// Tests for AstroBROT.FB_RADEC2HADEC (ICRS RA/Dec -> apparent hour angle / Dec; the block IAG50cm uses).
//
// GENERATED by AstroBROT/testing/gen_block_tests.py from testing/golden_blocks.py, do not edit the numbers by hand.
// Every golden case is checked against the Python port of the ST (1E-7 deg) and against erfa.atco13 as a great-circle
// separation on the (HA, Dec) sphere (2E-4 deg = 0.72 arcsec; the port is 0.2 to 0.4 arcsec away, mostly the diurnal
// aberration that the ST leaves out). The dut1 shift itself is also covered in FB_DUT1_Tests.
//
// Every call assigns all inputs: FB_RADEC2HADEC still writes its precessed and corrected position back into ra and dec
// (issue #8), so these tests must not rely on ra / dec surviving a call.
FUNCTION_BLOCK FB_RADEC2HADEC_Tests EXTENDS TcUnit.FB_TestSuite
VAR
END_VAR

Golden_Tenerife_2026();
Golden_Tenerife_low();
Golden_South_2010();
Golden_Dut1();
Golden_RA_Wrap();
Golden_Poles();
Golden_Near_The_Poles();
Right_Ascension_Is_Periodic();
Longitude_Is_Periodic();
Outputs_Stay_In_Range();
Time_Inputs_Are_Not_Modified();

METHOD PRIVATE CheckNear
VAR_INPUT
	fExpected	: LREAL;
	fActual	: LREAL;
	fDelta	: LREAL;
	sName	: STRING(255);
END_VAR
AssertEquals_LREAL(Expected := fExpected, Actual := fActual, Delta := fDelta, Message := sName);
END_METHOD

METHOD PRIVATE CheckAngle
VAR_INPUT
	fExpected	: LREAL;
	fActual	: LREAL;
	fDelta	: LREAL;
	sName	: STRING(255);
END_VAR
VAR
	fDiff	: LREAL;
END_VAR
// angles in degrees, compared modulo 360 so that 359.9999999 and -1.0E-7 are equal
fDiff := fActual - fExpected;
WHILE fDiff > 180.0 DO fDiff := fDiff - 360.0; END_WHILE
WHILE fDiff < -180.0 DO fDiff := fDiff + 360.0; END_WHILE
AssertEquals_LREAL(Expected := 0.0, Actual := fDiff, Delta := fDelta, Message := sName);
END_METHOD

METHOD PRIVATE CheckSeparation
VAR_INPUT
	fLon1	: LREAL;
	fLat1	: LREAL;
	fLon2	: LREAL;
	fLat2	: LREAL;
	fDelta	: LREAL;
	sName	: STRING(255);
END_VAR
VAR
	fD2r	: LREAL;
	fHalfDLat	: LREAL;
	fHalfDLon	: LREAL;
	fHav	: LREAL;
	fSep	: LREAL;
END_VAR
// great-circle separation of two positions (longitude, latitude in degrees) against a tolerance in degrees;
// a difference of longitudes is not a distance on the sky, this is (haversine formula)
fD2r := 0.017453292519943295;
fHalfDLat := (fLat2 - fLat1) * fD2r * 0.5;
fHalfDLon := (fLon2 - fLon1) * fD2r * 0.5;
fHav := SIN(fHalfDLat) * SIN(fHalfDLat) + COS(fLat1 * fD2r) * COS(fLat2 * fD2r) * SIN(fHalfDLon) * SIN(fHalfDLon);
fSep := 2.0 * ASIN(SQRT(LIMIT(0.0, fHav, 1.0))) / fD2r;
AssertEquals_LREAL(Expected := 0.0, Actual := fSep, Delta := fDelta, Message := sName);
END_METHOD

METHOD PRIVATE Golden_Tenerife_2026
VAR
	fb	: AstroBROT.FB_RADEC2HADEC;
END_VAR
TEST('Golden_Tenerife_2026');
fb(jd := 2461300.75, ra := 83.63, dec := 22.01, lon := -16.5, dut1 := 0.0);
CheckAngle(345.6575630310487, fb.ha_out, 1.0E-7, 'Tenerife_2026 ha');
CheckNear(22.02849232968123, fb.dec_out, 1.0E-7, 'Tenerife_2026 dec');
CheckSeparation(345.65746144326204, 22.028485286326138, fb.ha_out, fb.dec_out, 0.0002, 'Tenerife_2026 vs erfa');
TEST_FINISHED();
END_METHOD

METHOD PRIVATE Golden_Tenerife_low
VAR
	fb	: AstroBROT.FB_RADEC2HADEC;
END_VAR
TEST('Golden_Tenerife_low');
fb(jd := 2461300.75, ra := 130.0, dec := -10.0, lon := -16.5, dut1 := 0.0);
CheckAngle(299.37201176540054, fb.ha_out, 1.0E-7, 'Tenerife_low ha');
CheckNear(-10.091922210560911, fb.dec_out, 1.0E-7, 'Tenerife_low dec');
CheckSeparation(299.3719555337581, -10.091909866750818, fb.ha_out, fb.dec_out, 0.0002, 'Tenerife_low vs erfa');
TEST_FINISHED();
END_METHOD

METHOD PRIVATE Golden_South_2010
VAR
	fb	: AstroBROT.FB_RADEC2HADEC;
END_VAR
TEST('Golden_South_2010');
fb(jd := 2455197.5, ra := 312.5, dec := -47.3, lon := -70.7, dut1 := 0.0);
CheckAngle(77.17023586398261, fb.ha_out, 1.0E-7, 'South_2010 ha');
CheckNear(-47.26426875549772, fb.dec_out, 1.0E-7, 'South_2010 dec');
CheckSeparation(77.17019695311718, -47.26432489859199, fb.ha_out, fb.dec_out, 0.0002, 'South_2010 vs erfa');
TEST_FINISHED();
END_METHOD

METHOD PRIVATE Golden_Dut1
VAR
	fb	: AstroBROT.FB_RADEC2HADEC;
END_VAR
TEST('Golden_Dut1');
fb(jd := 2461300.75, ra := 83.63, dec := 22.01, lon := -16.5, dut1 := 0.9);
CheckAngle(345.6613233618934, fb.ha_out, 1.0E-7, 'Tenerife_dut1_plus ha');
CheckNear(22.02849232968123, fb.dec_out, 1.0E-7, 'Tenerife_dut1_plus dec');
CheckSeparation(345.66122170868215, 22.028485288193934, fb.ha_out, fb.dec_out, 0.0002, 'Tenerife_dut1_plus vs erfa');
fb(jd := 2461300.75, ra := 83.63, dec := 22.01, lon := -16.5, dut1 := -0.9);
CheckAngle(345.65380270020404, fb.ha_out, 1.0E-7, 'Tenerife_dut1_minus ha');
CheckNear(22.02849232968123, fb.dec_out, 1.0E-7, 'Tenerife_dut1_minus dec');
CheckSeparation(345.653701177839, 22.028485284458373, fb.ha_out, fb.dec_out, 0.0002, 'Tenerife_dut1_minus vs erfa');
TEST_FINISHED();
END_METHOD

METHOD PRIVATE Golden_RA_Wrap
VAR
	fb	: AstroBROT.FB_RADEC2HADEC;
END_VAR
TEST('Golden_RA_Wrap');
fb(jd := 2461300.75, ra := 0.0001, dec := 22.01, lon := -16.5, dut1 := 0.0);
CheckAngle(69.34278166497118, fb.ha_out, 1.0E-7, 'RA_wrap_low ha');
CheckNear(22.16156103752678, fb.dec_out, 1.0E-7, 'RA_wrap_low dec');
CheckSeparation(69.34272927043514, 22.16158906186533, fb.ha_out, fb.dec_out, 0.0002, 'RA_wrap_low vs erfa');
fb(jd := 2461300.75, ra := 359.9999, dec := 22.01, lon := -16.5, dut1 := 0.0);
CheckAngle(69.34298187519398, fb.ha_out, 1.0E-7, 'RA_wrap_high ha');
CheckNear(22.16156103790214, fb.dec_out, 1.0E-7, 'RA_wrap_high dec');
CheckSeparation(69.34292948093092, 22.161589062278132, fb.ha_out, fb.dec_out, 0.0002, 'RA_wrap_high vs erfa');
TEST_FINISHED();
END_METHOD

METHOD PRIVATE Golden_Poles
VAR
	fb	: AstroBROT.FB_RADEC2HADEC;
END_VAR
TEST('Golden_Poles');
fb(jd := 2461300.75, ra := 0.0, dec := 90.0, lon := -16.5, dut1 := 0.0);
CheckAngle(250.63644034864151, fb.ha_out, 1.0E-7, 'North_pole ha');
CheckNear(89.85080571177119, fb.dec_out, 1.0E-7, 'North_pole dec');
CheckSeparation(250.63721443708533, 89.8507228178902, fb.ha_out, fb.dec_out, 0.0002, 'North_pole vs erfa');
fb(jd := 2455197.5, ra := 0.0, dec := -90.0, lon := -70.7, dut1 := 0.0);
CheckAngle(29.9862312944732, fb.ha_out, 1.0E-7, 'South_pole ha');
CheckNear(-89.94820320442783, fb.dec_out, 1.0E-7, 'South_pole dec');
CheckSeparation(29.899988989677052, -89.94824504562501, fb.ha_out, fb.dec_out, 0.0002, 'South_pole vs erfa');
TEST_FINISHED();
END_METHOD

METHOD PRIVATE Golden_Near_The_Poles
VAR
	fb	: AstroBROT.FB_RADEC2HADEC;
END_VAR
TEST('Golden_Near_The_Poles');
fb(jd := 2461300.75, ra := 200.0, dec := 89.9, lon := -16.5, dut1 := 0.0);
CheckAngle(242.11458567841964, fb.ha_out, 1.0E-7, 'Near_north_pole ha');
CheckNear(89.75492331909197, fb.dec_out, 1.0E-7, 'Near_north_pole dec');
CheckSeparation(242.12047093980044, 89.75484732066303, fb.ha_out, fb.dec_out, 0.0002, 'Near_north_pole vs erfa');
fb(jd := 2455197.5, ra := 200.0, dec := -89.9, lon := -70.7, dut1 := 0.0);
CheckAngle(170.60136769350444, fb.ha_out, 1.0E-7, 'Near_south_pole ha');
CheckNear(-89.94559816252283, fb.dec_out, 1.0E-7, 'Near_south_pole dec');
CheckSeparation(170.55436891323328, -89.9455612839385, fb.ha_out, fb.dec_out, 0.0002, 'Near_south_pole vs erfa');
TEST_FINISHED();
END_METHOD

METHOD PRIVATE Right_Ascension_Is_Periodic
VAR
	fb	: AstroBROT.FB_RADEC2HADEC;
END_VAR
TEST('Right_Ascension_Is_Periodic');
// ra and ra +- 360 are the same position
fb(jd := 2461300.75, ra := -276.37, dec := 22.01, lon := -16.5);
CheckAngle(345.6575630310487, fb.ha_out, 1.0E-9, 'ra - 360 ha');
CheckNear(22.02849232968123, fb.dec_out, 1.0E-9, 'ra - 360 dec');
fb(jd := 2461300.75, ra := 443.63, dec := 22.01, lon := -16.5);
CheckAngle(345.6575630310487, fb.ha_out, 1.0E-9, 'ra + 360 ha');
CheckNear(22.02849232968123, fb.dec_out, 1.0E-9, 'ra + 360 dec');
TEST_FINISHED();
END_METHOD

METHOD PRIVATE Longitude_Is_Periodic
VAR
	fb	: AstroBROT.FB_RADEC2HADEC;
END_VAR
TEST('Longitude_Is_Periodic');
// lon and lon +- 360 are the same place
fb(jd := 2461300.75, ra := 83.63, dec := 22.01, lon := 343.5);
CheckAngle(345.6575630310487, fb.ha_out, 1.0E-9, 'lon + 360 ha');
fb(jd := 2461300.75, ra := 83.63, dec := 22.01, lon := -376.5);
CheckAngle(345.6575630310487, fb.ha_out, 1.0E-9, 'lon - 360 ha');
TEST_FINISHED();
END_METHOD

METHOD PRIVATE Outputs_Stay_In_Range
VAR
	fb	: AstroBROT.FB_RADEC2HADEC;
	i	: INT;
	fRa	: LREAL;
END_VAR
TEST('Outputs_Stay_In_Range');
// a sweep over the whole RA circle and the declinations up to and including the poles
FOR i := 0 TO 8 DO
	fRa := 45.0 * i;
	fb(jd := 2461300.75, ra := fRa, dec := 90.0, lon := -16.5);
	AssertTrue(Condition := fb.ha_out >= 0.0 AND fb.ha_out < 360.0 AND fb.dec_out <= 90.0 AND fb.dec_out >= -90.0, Message := 'ra sweep at dec +90 stays in range');
	fb(jd := 2461300.75, ra := fRa, dec := -90.0, lon := -16.5);
	AssertTrue(Condition := fb.ha_out >= 0.0 AND fb.ha_out < 360.0 AND fb.dec_out <= 90.0 AND fb.dec_out >= -90.0, Message := 'ra sweep at dec -90 stays in range');
	fb(jd := 2461300.75, ra := fRa, dec := 0.0, lon := -16.5);
	AssertTrue(Condition := fb.ha_out >= 0.0 AND fb.ha_out < 360.0 AND fb.dec_out <= 90.0 AND fb.dec_out >= -90.0, Message := 'ra sweep at dec 0 stays in range');
END_FOR
TEST_FINISHED();
END_METHOD

METHOD PRIVATE Time_Inputs_Are_Not_Modified
VAR
	fb	: AstroBROT.FB_RADEC2HADEC;
END_VAR
TEST('Time_Inputs_Are_Not_Modified');
fb(jd := 2461300.75, ra := 83.63, dec := 22.01, lon := -16.5, dut1 := 0.5);
CheckNear(2461300.75, fb.jd, 0.0, 'jd unchanged');
CheckNear(-16.5, fb.lon, 0.0, 'lon unchanged');
CheckNear(0.5, fb.dut1, 0.0, 'dut1 unchanged');
TEST_FINISHED();
END_METHOD

END_FUNCTION_BLOCK

(* stored: Version 1.1.0.1, ProductVersion 3.1.4024.15
   POU FB_RADEC2HADEC_Tests: Id {5b5d6534-9c2d-57c7-bcb9-f8625c087574}, SpecialFunc None
   Method CheckNear: Id {dafe04a7-9323-5fd0-82ce-90cd84bf0880}
   Method CheckAngle: Id {c1e9619b-4370-558b-b594-843ebe494fe2}
   Method CheckSeparation: Id {cb9fb004-4f5b-5971-97da-e3f6e06912e3}
   Method Golden_Tenerife_2026: Id {7eae40f9-c372-5220-a298-4c0c8ecf1e82}
   Method Golden_Tenerife_low: Id {3989c102-b65f-5568-8831-c0fd4a1e5552}
   Method Golden_South_2010: Id {17bce24d-8ec4-5584-b76f-f0b3efe5c72b}
   Method Golden_Dut1: Id {bada3be5-be41-559a-b6c9-17fb6156b95f}
   Method Golden_RA_Wrap: Id {309e2cba-c173-53f3-b463-980b0dbebe87}
   Method Golden_Poles: Id {22c3d7b4-897a-52c2-95c5-8821aec1568e}
   Method Golden_Near_The_Poles: Id {a2624210-469b-5a8e-bc6f-39dd853ec614}
   Method Right_Ascension_Is_Periodic: Id {630c859c-0151-5c52-8af6-f13b5c6be800}
   Method Longitude_Is_Periodic: Id {6721f928-dce0-54b5-9ec3-99fa33cf5532}
   Method Outputs_Stay_In_Range: Id {180e42aa-f9c3-5697-8eaa-001a29a46c42}
   Method Time_Inputs_Are_Not_Modified: Id {2dde0a0e-4033-542e-a641-d61f54ee417c} *)
